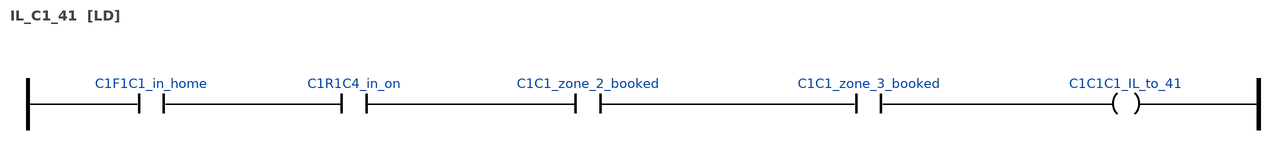
(* LD diagram, written out as Structured Text *)
C1C1C1_IL_to_41 := C1F1C1_in_home AND C1R1C4_in_on AND C1C1_zone_2_booked AND C1C1_zone_3_booked;
END_PROGRAM

PROGRAM IL_C1C2C1_PART_IN_POSITION
  VAR_EXTERNAL
    C1C2_zone_1_booked : BOOL := false;
    C1C2C1_IL_to_part_in_position : BOOL := false;
  END_VAR

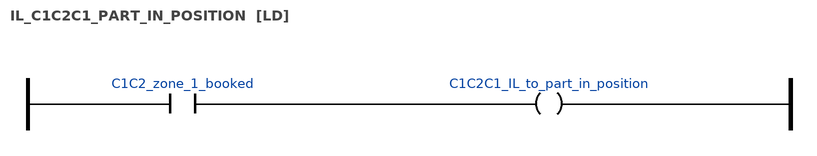
(* LD diagram, written out as Structured Text *)
C1C2C1_IL_to_part_in_position := C1C2_zone_1_booked;
END_PROGRAM

PROGRAM IL_C1C2C1_POSITION_EMPTY
  VAR_EXTERNAL
    C1C2C1_IL_to_part_in_position : BOOL := false;
  END_VAR

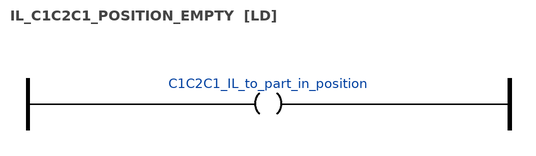
(* LD diagram, written out as Structured Text *)
C1C2C1_IL_to_part_in_position := TRUE;
END_PROGRAM

PROGRAM IL_F1C1_HOME_POS
  VAR_EXTERNAL
    C1F1C2_in_unlocked : BOOL := false;
    C1F1C4_in_off : BOOL := false;
    C1F1C3_in_close : BOOL := false;
    C1F1C4_in_on : BOOL := false;
    Op_24_start : BOOL := false;
    C1F1C3_in_open : BOOL := false;
    C1F1C1_IL_to_home : BOOL := false;
  END_VAR

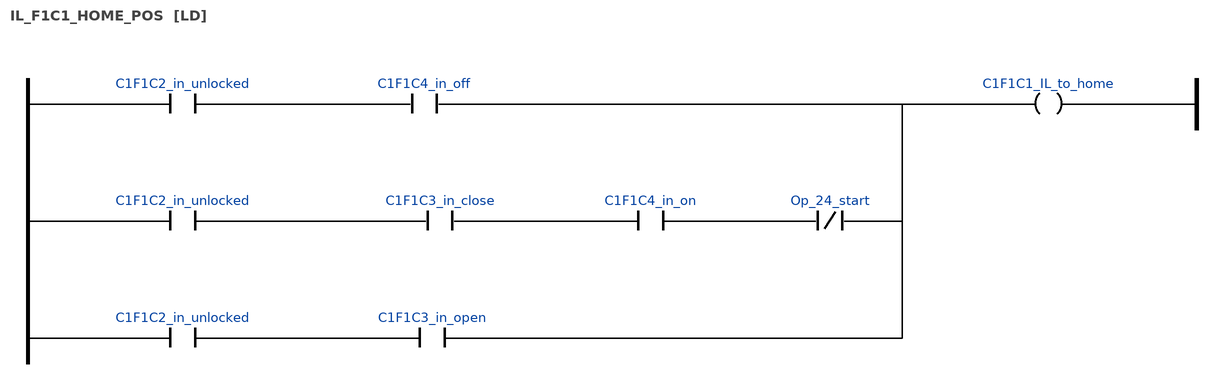
(* LD diagram, written out as Structured Text *)
C1F1C1_IL_to_home := C1F1C2_in_unlocked AND (C1F1C4_in_off OR C1F1C3_in_close AND C1F1C4_in_on AND NOT Op_24_start OR C1F1C3_in_open);
END_PROGRAM

PROGRAM IL_F1C1_WORK_POS
  VAR_EXTERNAL
    C1F1C2_in_unlocked : BOOL := false;
    C1F1C4_in_off : BOOL := false;
    C1F1_zone_2_booked : BOOL := false;
    Op_21_start : BOOL := false;
    Op_21_end : BOOL := false;
    C1F1C4_in_on : BOOL := false;
    C1C1C1_in_empty : BOOL := false;
    C1F1C1_to_work_pos_started : BOOL := false;
    C1F1_zone_3_booked : BOOL := false;
    C1C1C1_in_unprocessed : BOOL := false;
    Op_24_start : BOOL := false;
    C1F1C1_IL_to_work_pos : BOOL := false;
  END_VAR

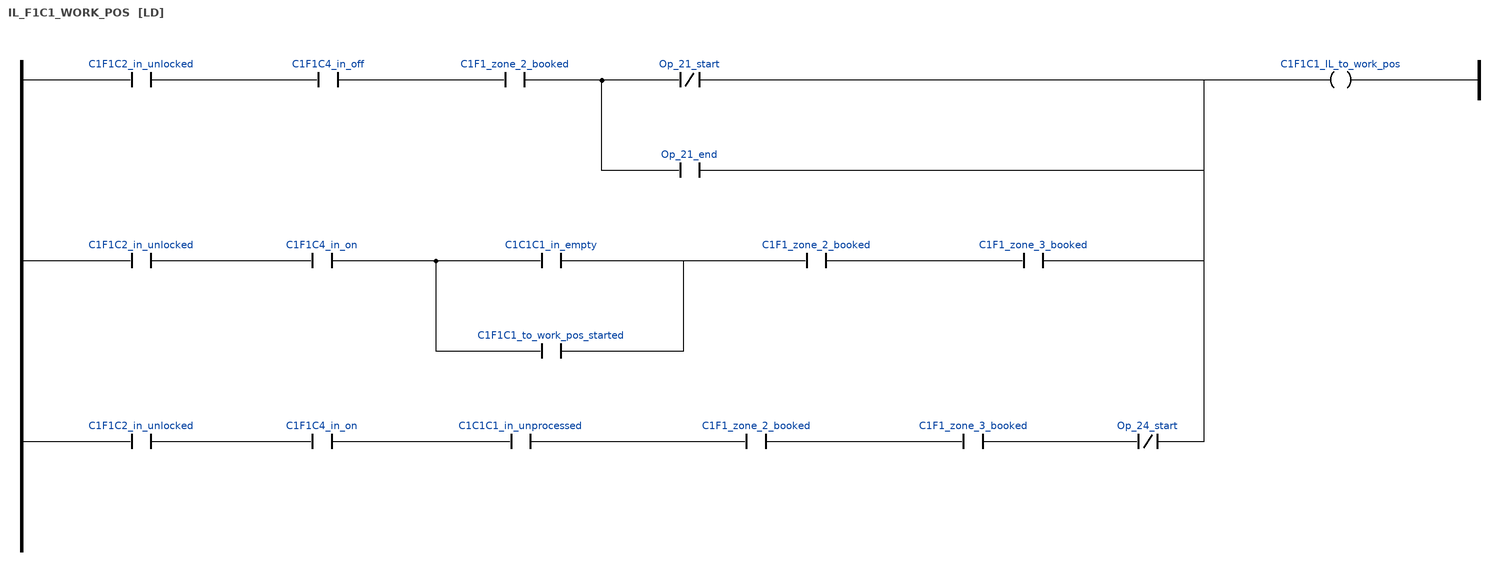
(* LD diagram, written out as Structured Text *)
C1F1C1_IL_to_work_pos := C1F1C2_in_unlocked AND (C1F1C4_in_off AND C1F1_zone_2_booked AND NOT Op_21_start OR C1F1C4_in_off AND C1F1_zone_2_booked AND Op_21_end OR C1F1C4_in_on AND (C1C1C1_in_empty OR C1F1C1_to_work_pos_started) AND C1F1_zone_2_booked AND C1F1_zone_3_booked OR C1F1C4_in_on AND C1C1C1_in_unprocessed AND C1F1_zone_2_booked AND C1F1_zone_3_booked AND NOT Op_24_start);
END_PROGRAM

PROGRAM IL_F1C2_LOCKED
  VAR_EXTERNAL
    C1F1C1_in_home : BOOL := false;
    C1F1C1_in_work_pos : BOOL := false;
    C1F1C2_IL_to_locked : BOOL := false;
  END_VAR

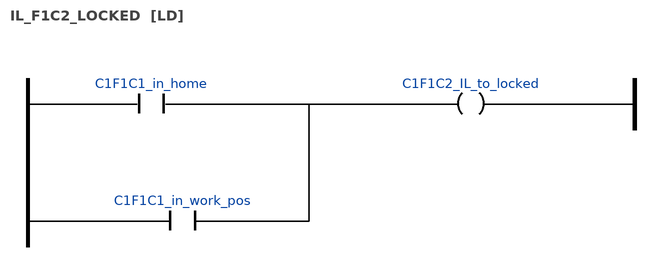
(* LD diagram, written out as Structured Text *)
C1F1C2_IL_to_locked := C1F1C1_in_home OR C1F1C1_in_work_pos;
END_PROGRAM

PROGRAM IL_F1C2_UNLOCKED
  VAR_EXTERNAL
    C1F1C2_IL_to_unlocked : BOOL := false;
  END_VAR

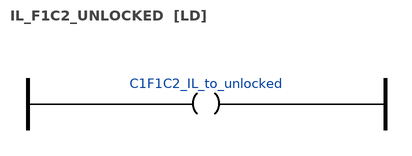
(* LD diagram, written out as Structured Text *)
C1F1C2_IL_to_unlocked := TRUE;
END_PROGRAM

PROGRAM IL_F1C3_CLOSED
  VAR_EXTERNAL
    C1F1C3_IL_to_closed : BOOL := false;
  END_VAR

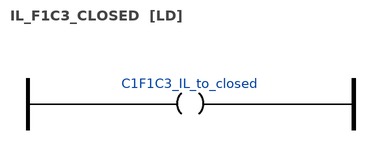
(* LD diagram, written out as Structured Text *)
C1F1C3_IL_to_closed := TRUE;
END_PROGRAM

PROGRAM IL_F1C3_OPEN
  VAR_EXTERNAL
    C1F1C1_in_home : BOOL := false;
    C1F1C1_in_work_pos : BOOL := false;
    C1F1C4_in_off : BOOL := false;
    C1F1C4_in_on : BOOL := false;
    Op_24_start : BOOL := false;
    Op_24_end : BOOL := false;
    C1F1C3_IL_to_open : BOOL := false;
  END_VAR

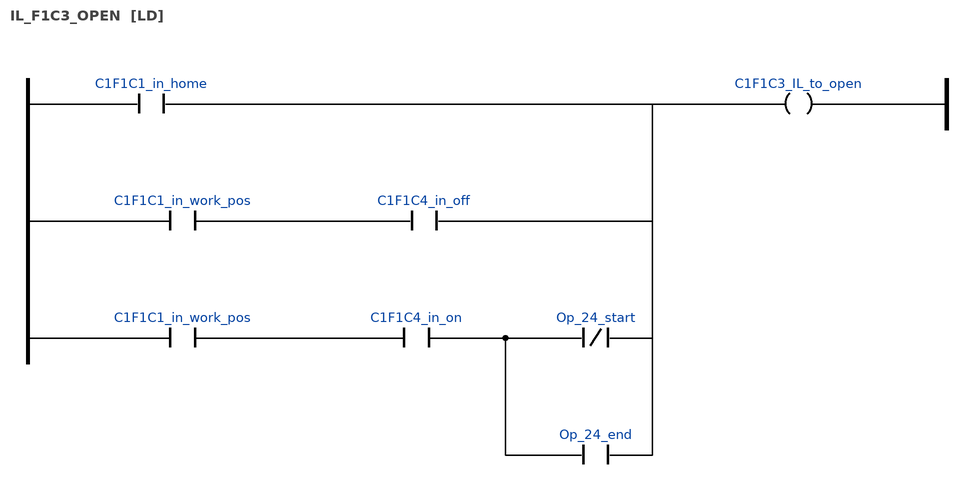
(* LD diagram, written out as Structured Text *)
C1F1C3_IL_to_open := C1F1C1_in_home OR C1F1C1_in_work_pos AND C1F1C4_in_off OR C1F1C1_in_work_pos AND C1F1C4_in_on AND NOT Op_24_start OR C1F1C1_in_work_pos AND C1F1C4_in_on AND Op_24_end;
END_PROGRAM

PROGRAM IL_R1_21
  VAR_EXTERNAL
    C1R1C1_in_open : BOOL := false;
    C1R1C2_in_off : BOOL := false;
    C1C2C1_in_part_in_position : BOOL := false;
    C1R1_zone_1_booked : BOOL := false;
    C1C2C1_in_position_empty : BOOL := false;
    C1R1C1R1_IL_to_21 : BOOL := false;
  END_VAR

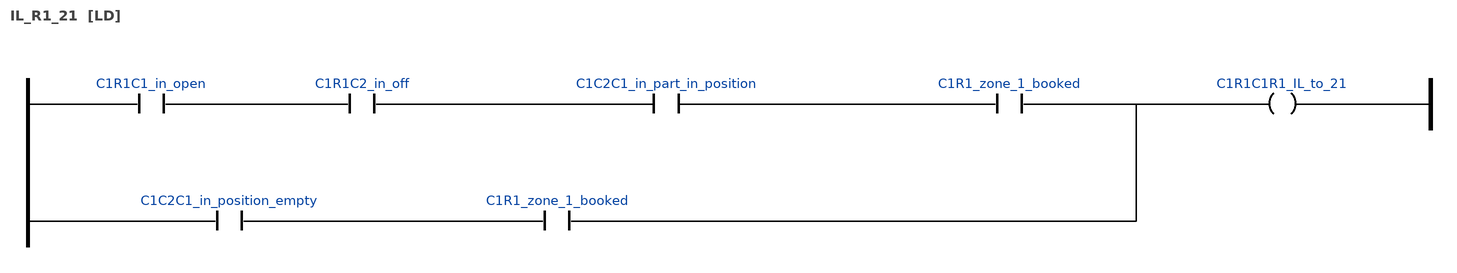
(* LD diagram, written out as Structured Text *)
C1R1C1R1_IL_to_21 := C1R1C1_in_open AND C1R1C2_in_off AND C1C2C1_in_part_in_position AND C1R1_zone_1_booked OR C1C2C1_in_position_empty AND C1R1_zone_1_booked;
END_PROGRAM

PROGRAM IL_R1_22
  VAR_EXTERNAL
    C1F1C1_in_home : BOOL := false;
    C1F1C2_in_locked : BOOL := false;
    C1F1C3_in_open : BOOL := false;
    C1F1C4_in_off : BOOL := false;
    C1R1_Op22_started : BOOL := false;
    C1R1_zone_2_booked : BOOL := false;
    C1R1C1R1_IL_to_22 : BOOL := false;
  END_VAR

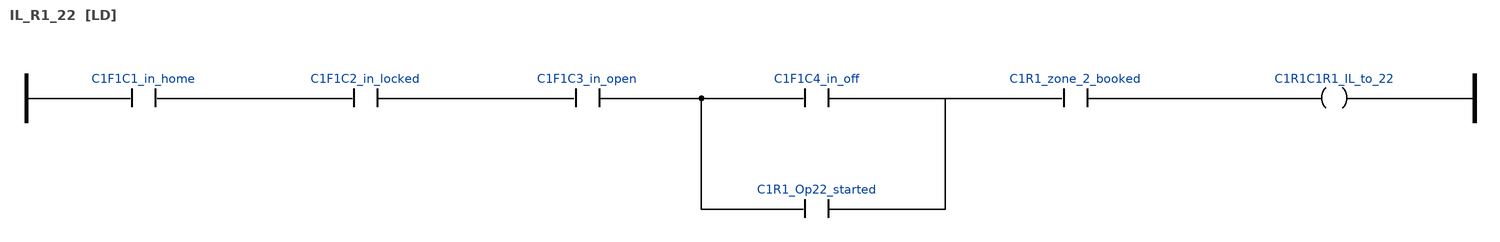
(* LD diagram, written out as Structured Text *)
C1R1C1R1_IL_to_22 := C1F1C1_in_home AND C1F1C2_in_locked AND C1F1C3_in_open AND (C1F1C4_in_off OR C1R1_Op22_started) AND C1R1_zone_2_booked;
END_PROGRAM

PROGRAM IL_R1_23
  VAR_EXTERNAL
    C1R1_zone_2_booked : BOOL := false;
    C1R1C1R1_IL_to_23 : BOOL := false;
  END_VAR

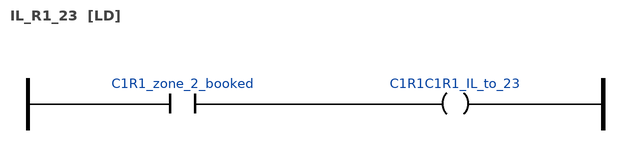
(* LD diagram, written out as Structured Text *)
C1R1C1R1_IL_to_23 := C1R1_zone_2_booked;
END_PROGRAM

PROGRAM IL_R1_24
  VAR_EXTERNAL
    C1C1C1_in_empty : BOOL := false;
    C1F1C1_in_home : BOOL := false;
    C1R1_zone_3_booked : BOOL := false;
    C1C1C1_in_unprocessed : BOOL := false;
    C1F1C1_in_work_pos : BOOL := false;
    C1F1C2_in_locked : BOOL := false;
    C1F1C3_in_open : BOOL := false;
    C1F1C4_in_off : BOOL := false;
    C1F1C3_in_close : BOOL := false;
    C1F1C4_in_on : BOOL := false;
    C1R1C1R1_IL_to_24 : BOOL := false;
  END_VAR

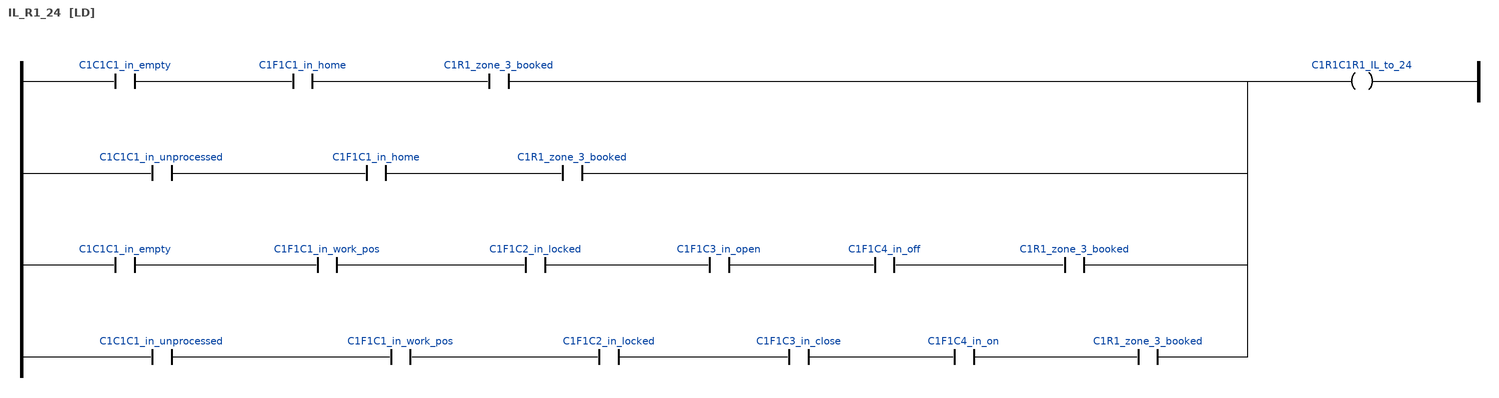
(* LD diagram, written out as Structured Text *)
C1R1C1R1_IL_to_24 := C1C1C1_in_empty AND C1F1C1_in_home AND C1R1_zone_3_booked OR C1C1C1_in_unprocessed AND C1F1C1_in_home AND C1R1_zone_3_booked OR C1C1C1_in_empty AND C1F1C1_in_work_pos AND C1F1C2_in_locked AND C1F1C3_in_open AND C1F1C4_in_off AND C1R1_zone_3_booked OR C1C1C1_in_unprocessed AND C1F1C1_in_work_pos AND C1F1C2_in_locked AND C1F1C3_in_close AND C1F1C4_in_on AND C1R1_zone_3_booked;
END_PROGRAM

PROGRAM CC
  VAR_EXTERNAL
    C1C2C1_in_position_empty : BOOL := false;
    C1C2C2_in_off : BOOL := false;
    C1C2C1_in_part_in_position : BOOL := false;
    C1C2C2_in_on : BOOL := false;
    C1R1_in_inital : BOOL := false;
    C1F1C1_in_home : BOOL := false;
    C1F1C2_in_locked : BOOL := false;
    C1F1C3_in_open : BOOL := false;
    C1F1C4_in_off : BOOL := false;
    C1H1C1_in_normal : BOOL := false;
    CC_B : BOOL := false;
    C1H1C1_in_empty : BOOL := false;
    C1C1C1_in_processed : BOOL := false;
    CC_A : BOOL := false;
    C1_init_position : BOOL := false;
    C1_auto : BOOL := false;
    Start_COPs : BOOL := false;
    COP_C1C1_A_done : BOOL := false;
    COP_C1C2_A_done : BOOL := false;
    COP_C1F1_A_done : BOOL := false;
    COP_C1R1_A_done : BOOL := false;
    All_COP_Done_CC_A : BOOL := false;
    COP_C1C1_B_done : BOOL := false;
    COP_C1C2_B_done : BOOL := false;
    COP_C1F1_B_done : BOOL := false;
    All_COP_Done_CC_B : BOOL := false;
    Op_10_end : BOOL := false;
    Op_11_end : BOOL := false;
    Op_12_end : BOOL := false;
    C1R1_Op20_done : BOOL := false;
    C1R1_Op21_done : BOOL := false;
    C1R1_Op22_done : BOOL := false;
    C1R1_Op23_done : BOOL := false;
    C1R1_Op24_done : BOOL := false;
    Op_30_end : BOOL := false;
    Op_31_end : BOOL := false;
    Op_32_end : BOOL := false;
    Op_33_end : BOOL := false;
    Op_34_end : BOOL := false;
    C1C1_Op40_done : BOOL := false;
    C1C1_Op41_done : BOOL := false;
    C1C1_Op42_done : BOOL := false;
  END_VAR
  VAR  (* added by the conversion: wires and edge detectors of the diagram *)
    _OR45_OUT : BOOL;
  END_VAR

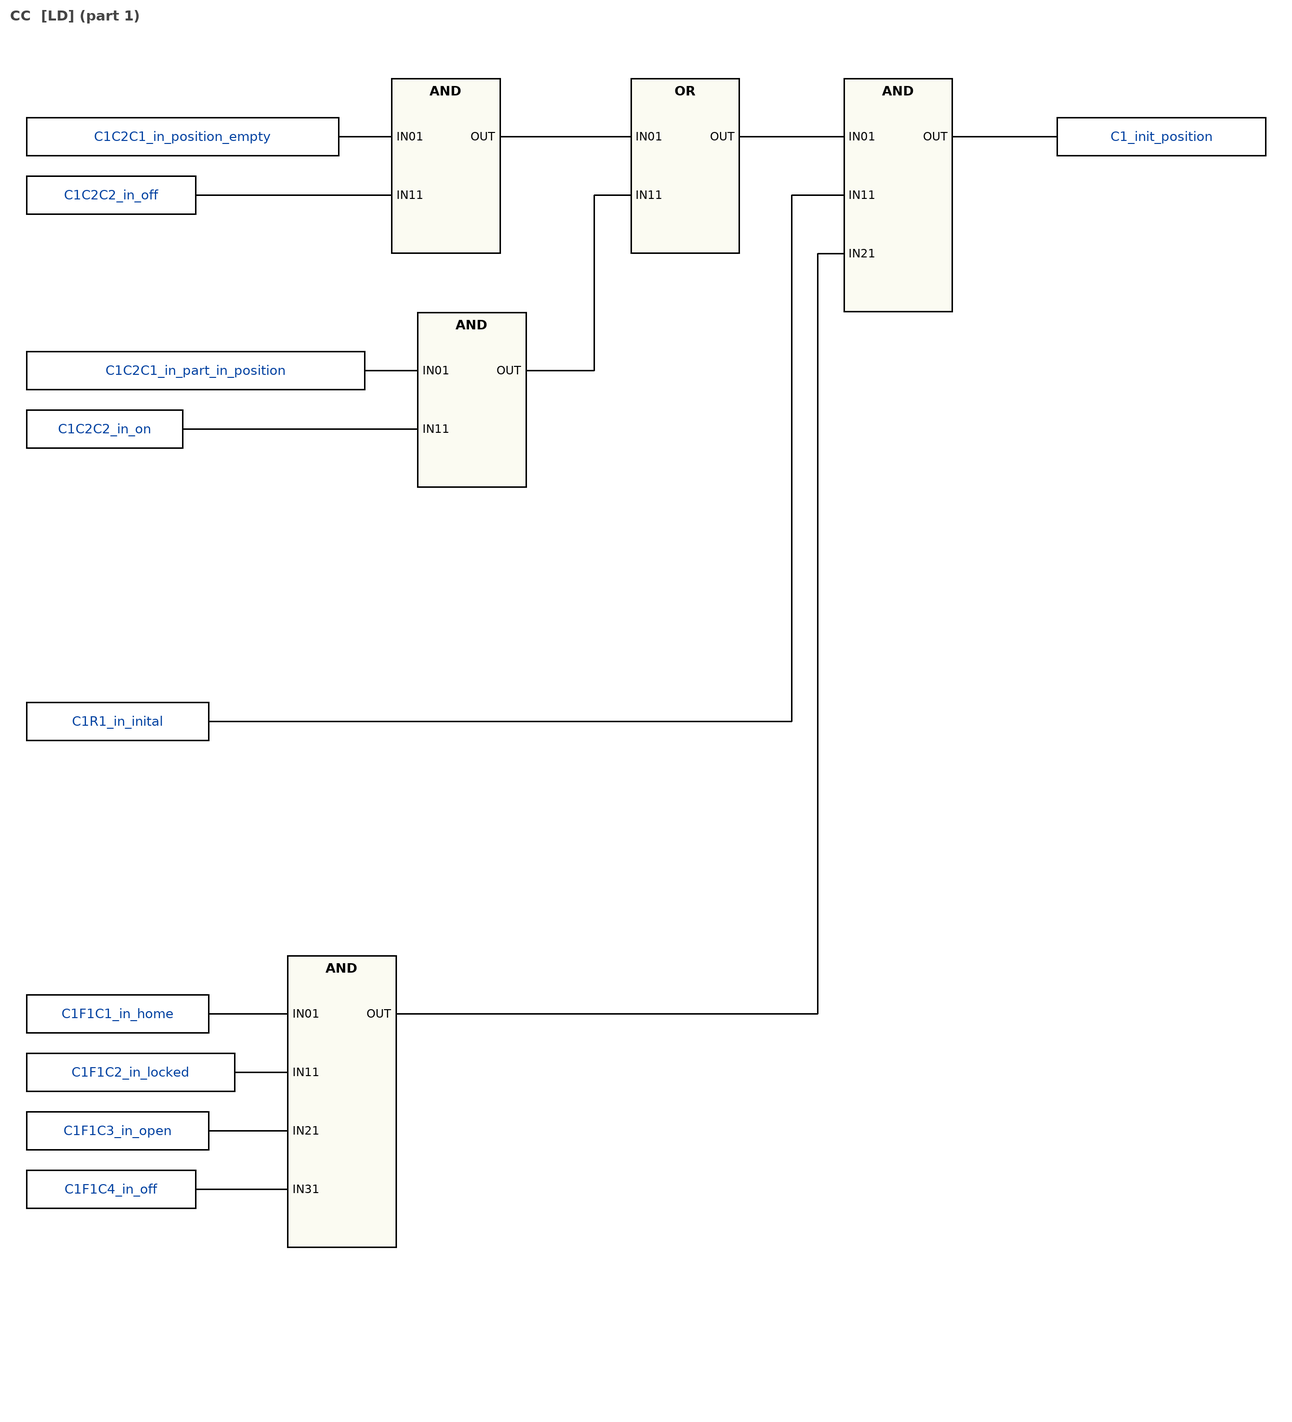
(* LD diagram, written out as Structured Text *)
C1_init_position := (C1C2C1_in_position_empty AND C1C2C2_in_off OR C1C2C1_in_part_in_position AND C1C2C2_in_on) AND C1R1_in_inital AND C1F1C1_in_home AND C1F1C2_in_locked AND C1F1C3_in_open AND C1F1C4_in_off;
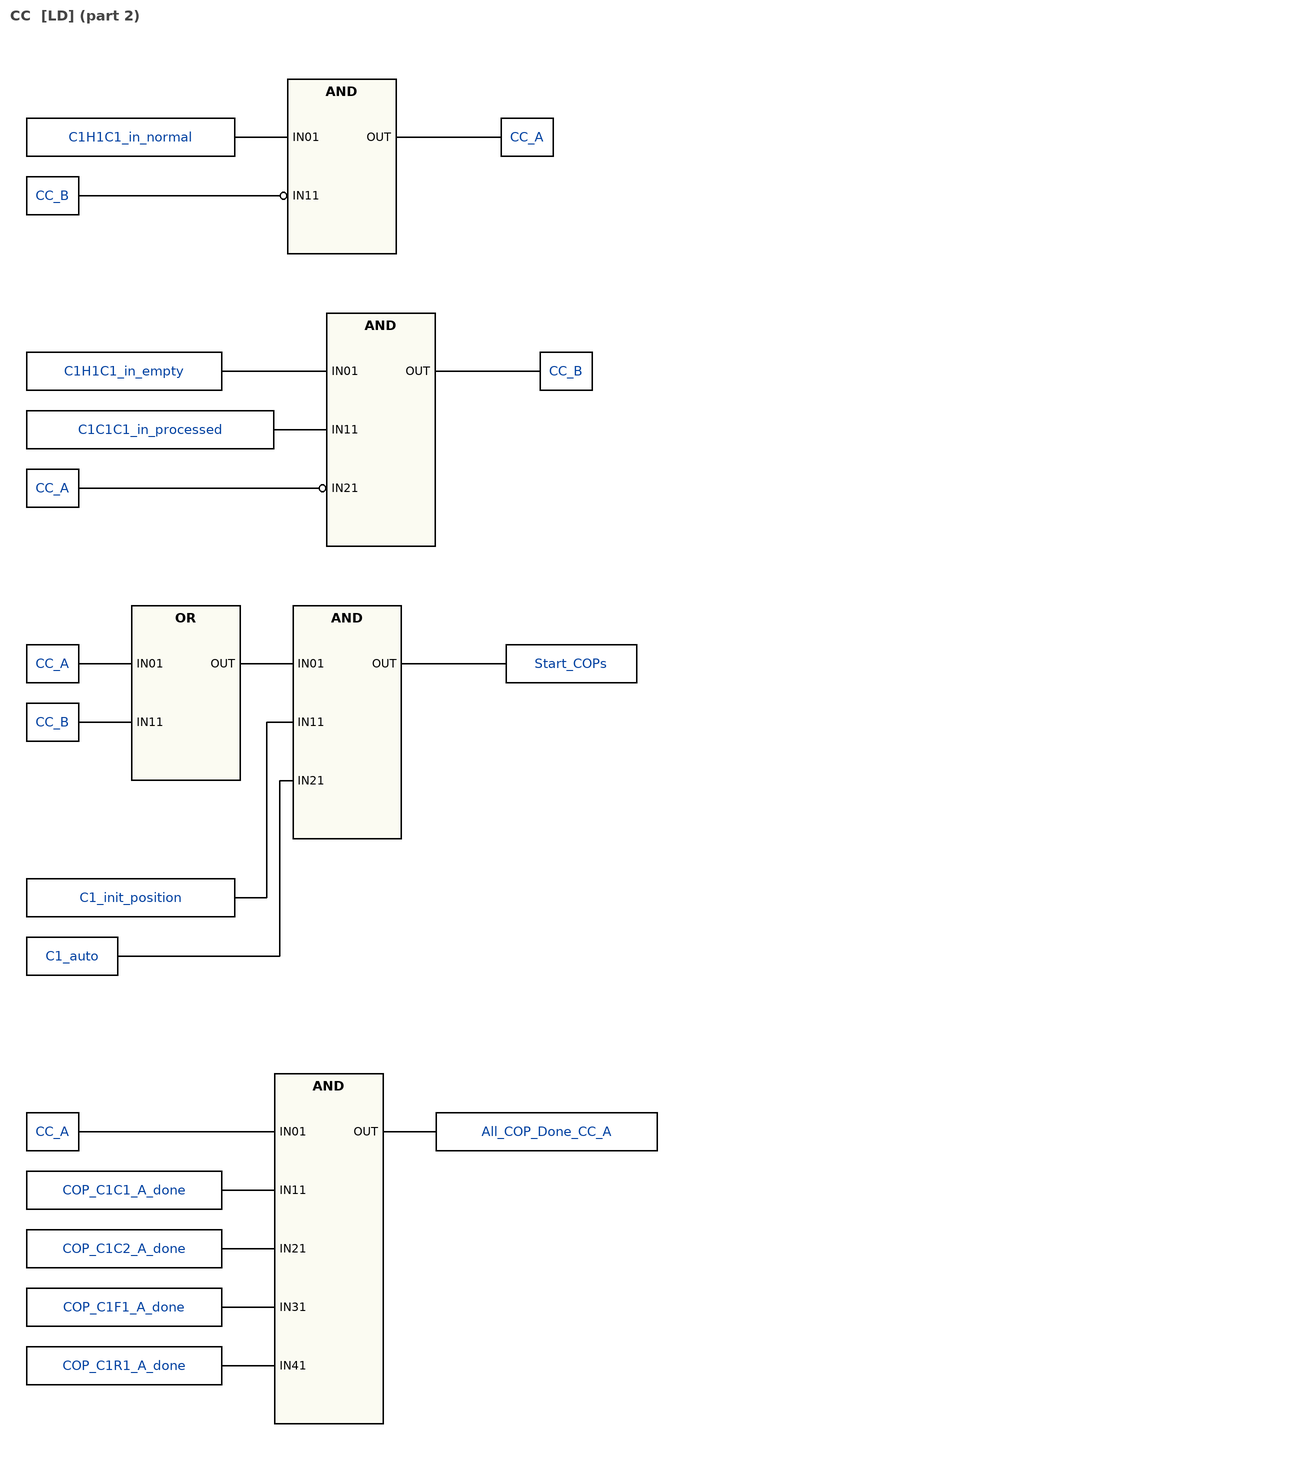
CC_A := C1H1C1_in_normal AND NOT CC_B;
CC_B := C1H1C1_in_empty AND C1C1C1_in_processed AND NOT CC_A;
Start_COPs := (CC_A OR CC_B) AND C1_init_position AND C1_auto;
All_COP_Done_CC_A := CC_A AND COP_C1C1_A_done AND COP_C1C2_A_done AND COP_C1F1_A_done AND COP_C1R1_A_done;
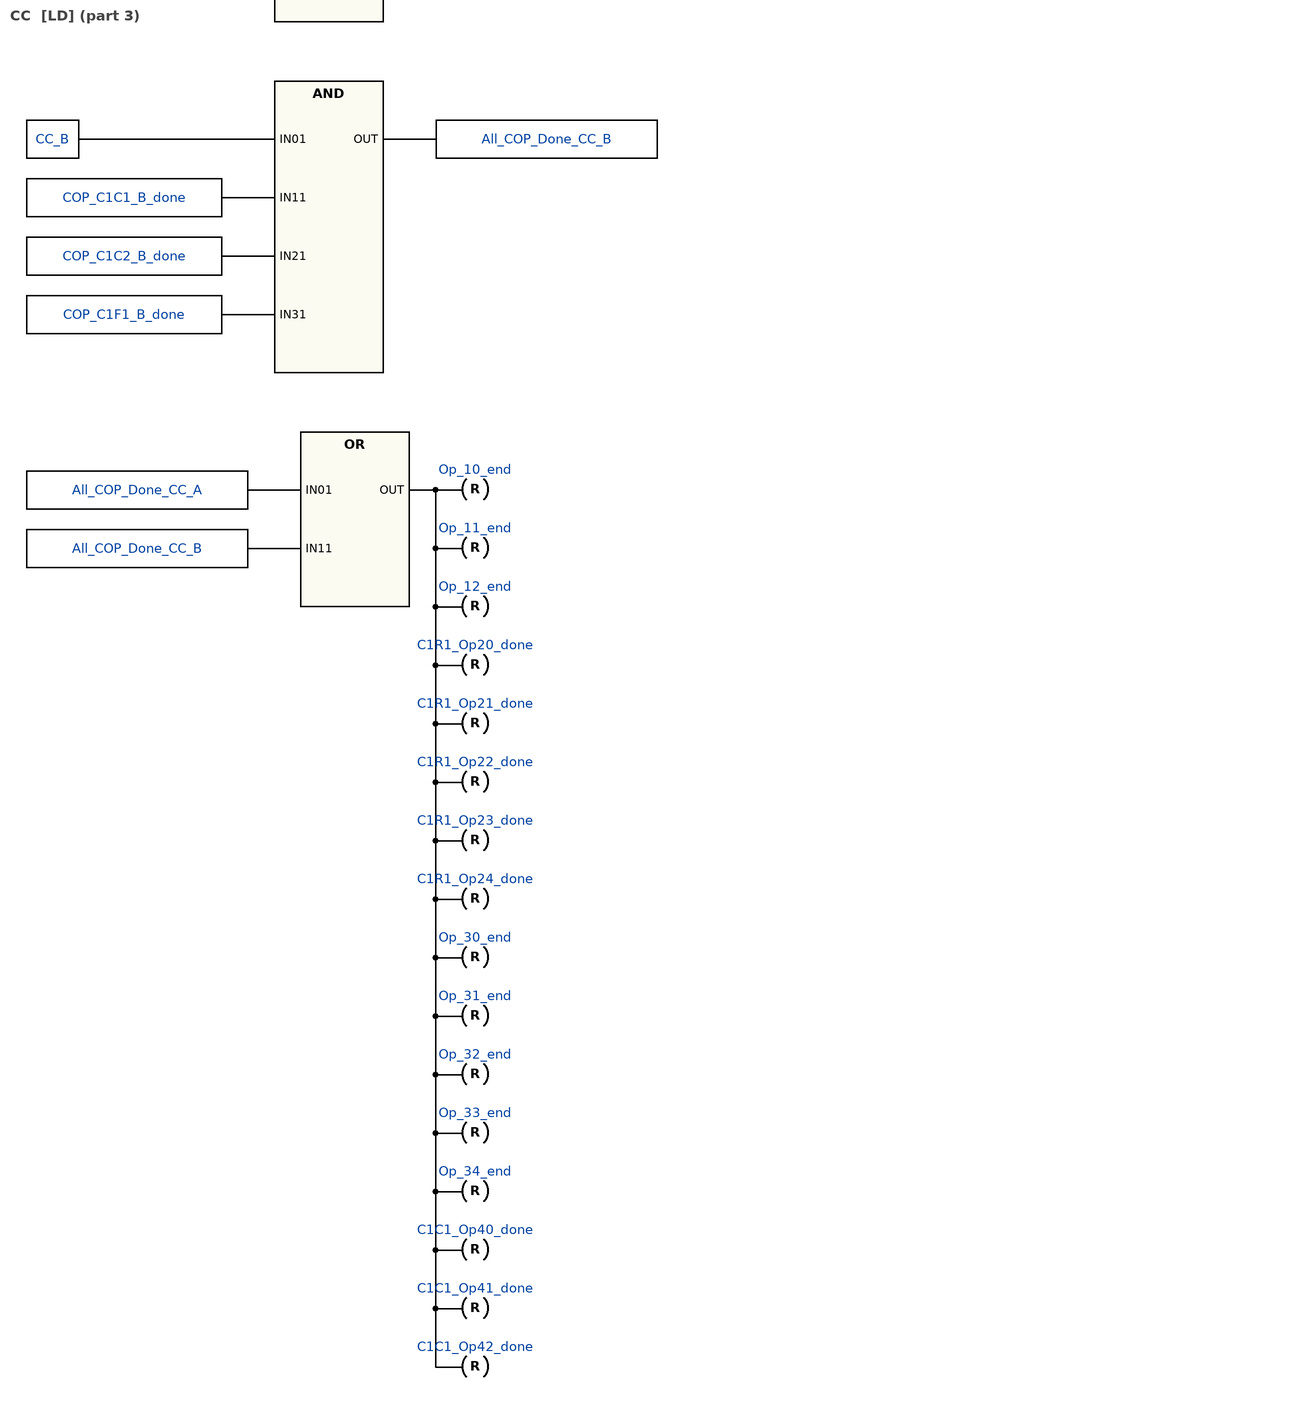
All_COP_Done_CC_B := CC_B AND COP_C1C1_B_done AND COP_C1C2_B_done AND COP_C1F1_B_done;
_OR45_OUT := All_COP_Done_CC_A OR All_COP_Done_CC_B;
IF _OR45_OUT THEN Op_10_end := FALSE; END_IF;
IF _OR45_OUT THEN Op_11_end := FALSE; END_IF;
IF _OR45_OUT THEN Op_12_end := FALSE; END_IF;
IF _OR45_OUT THEN C1R1_Op20_done := FALSE; END_IF;
IF _OR45_OUT THEN C1R1_Op21_done := FALSE; END_IF;
IF _OR45_OUT THEN C1R1_Op22_done := FALSE; END_IF;
IF _OR45_OUT THEN C1R1_Op23_done := FALSE; END_IF;
IF _OR45_OUT THEN C1R1_Op24_done := FALSE; END_IF;
IF _OR45_OUT THEN Op_30_end := FALSE; END_IF;
IF _OR45_OUT THEN Op_31_end := FALSE; END_IF;
IF _OR45_OUT THEN Op_32_end := FALSE; END_IF;
IF _OR45_OUT THEN Op_33_end := FALSE; END_IF;
IF _OR45_OUT THEN Op_34_end := FALSE; END_IF;
IF _OR45_OUT THEN C1C1_Op40_done := FALSE; END_IF;
IF _OR45_OUT THEN C1C1_Op41_done := FALSE; END_IF;
IF _OR45_OUT THEN C1C1_Op42_done := FALSE; END_IF;
END_PROGRAM

CONFIGURATION Example_factory002
  RESOURCE Example_cell002 ON PLC
    VAR_GLOBAL
      Op_10_start : BOOL := false;
      C1C2C1_in_position_empty : BOOL := false;
      C1C2C2_in_off : BOOL := false;
      Op_10_end : BOOL := false;
      C1C2C1_in_part_in_position : BOOL := false;
      C1C2C2_in_on : BOOL := false;
      Op_11_start : BOOL := false;
      TRUE_VAR : BOOL := true;
      C1C2_book_zone_1 : BOOL := false;
      C1C2_zone_1_booked : BOOL := false;
      C1C2C1_goto_part_in_position : BOOL := false;
      C1C2C2_goto_on : BOOL := false;
      C1C2_unbook_zone_1 : BOOL := false;
      Op_11_end : BOOL := false;
      Op_12_start : BOOL := false;
      C1C2C1_goto_position_empty : BOOL := false;
      C1C2C2_goto_off : BOOL := false;
      Op_12_end : BOOL := false;
      C1R1_Op20_exe_start : BOOL := false;
      C1R1_in_inital : BOOL := false;
      C1R1_Op20_exe : BOOL := false;
      C1R1_Op20_done : BOOL := false;
      C1R1_Op21_exe_start : BOOL := false;
      C1R1_book_zone_1 : BOOL := false;
      C1R1_zone_1_booked : BOOL := false;
      C1R1_Op21_exe : BOOL := false;
      C1R1_Op21_done : BOOL := false;
      C1R1_unbook_zone_1 : BOOL := false;
      C1R1_Op22_exe_start : BOOL := false;
      C1R1_Op22_exe : BOOL := false;
      C1R1_Op22_done : BOOL := false;
      C1R1_Op23_exe_start : BOOL := false;
      C1R1_book_zone_2 : BOOL := false;
      C1R1_zone_2_booked : BOOL := false;
      C1R1_Op23_exe : BOOL := false;
      C1R1_Op23_done : BOOL := false;
      C1R1_unbook_zone_2 : BOOL := false;
      C1R1_Op24_exe_start : BOOL := false;
      C1R1_book_zone_3 : BOOL := false;
      C1R1_zone_3_booked : BOOL := false;
      C1R1_Op24_exe : BOOL := false;
      C1R1_Op24_done : BOOL := false;
      C1R1_unbook_zone_3 : BOOL := false;
      Op_30_start : BOOL := false;
      C1F1C1_in_home : BOOL := false;
      C1F1C2_in_locked : BOOL := false;
      C1F1C3_in_open : BOOL := false;
      C1F1C4_in_off : BOOL := false;
      Op_30_end : BOOL := false;
      Op_31_start : BOOL := false;
      Op_31_end : BOOL := false;
      Op_32_start : BOOL := false;
      C1F1C1_goto_home : BOOL := false;
      C1F1C2_goto_locked : BOOL := false;
      C1F1C3_goto_close : BOOL := false;
      C1F1C4_goto_on : BOOL := false;
      C1F1C3_in_close : BOOL := false;
      C1F1C4_in_on : BOOL := false;
      Op_32_end : BOOL := false;
      Op_33_start : BOOL := false;
      C1F1C2_goto_unlocked : BOOL := false;
      C1F1_book_zone_2 : BOOL := false;
      C1F1_book_zone_3 : BOOL := false;
      C1F1C2_in_unlocked : BOOL := false;
      C1F1_zone_2_booked : BOOL := false;
      C1F1_zone_3_booked : BOOL := false;
      C1F1C1_goto_work_pos : BOOL := false;
      C1F1C1_in_work_pos : BOOL := false;
      C1F1_unbook_zone_3 : BOOL := false;
      Op_33_end : BOOL := false;
      Op_34_start : BOOL := false;
      C1F1C3_goto_open : BOOL := false;
      C1F1C4_goto_off : BOOL := false;
      C1F1_unbook_zone_2 : BOOL := false;
      Op_34_end : BOOL := false;
      C1C1_Op40_exe_start : BOOL := false;
      C1C1_Op40_done : BOOL := false;
      C1C1_Op41_exe_start : BOOL := false;
      C1C1_book_zone_2 : BOOL := false;
      C1C1_book_zone_3 : BOOL := false;
      C1C1_zone_2_booked : BOOL := false;
      C1C1_zone_3_booked : BOOL := false;
      C1C1C1_goto_unprocessed : BOOL := false;
      C1C1C1_in_unprocessed : BOOL := false;
      C1C1_unbook_zone_2 : BOOL := false;
      C1C1_unbook_zone_3 : BOOL := false;
      C1C1_Op41_done : BOOL := false;
      C1C1_Op42_exe_start : BOOL := false;
      C1C1C1_goto_processed : BOOL := false;
      C1C1C1_in_processed : BOOL := false;
      C1C1_Op42_done : BOOL := false;
      Start_COPs : BOOL := false;
      CC_A : BOOL := false;
      COP_C1C1_A_done : BOOL := false;
      All_COP_Done_CC_A : BOOL := false;
      CC_B : BOOL := false;
      C1C1_Op43_exe_start : BOOL := false;
      C1C1_Op43_done : BOOL := false;
      COP_C1C1_B_done : BOOL := false;
      All_COP_Done_CC_B : BOOL := false;
      COP_C1C2_A_done : BOOL := false;
      COP_C1C2_B_done : BOOL := false;
      COP_C1F1_A_done : BOOL := false;
      COP_C1F1_B_done : BOOL := false;
      COP_C1R1_A_done : BOOL := false;
      C1R1_Op20_IL : BOOL := false;
      C1R1_Op20_started : BOOL := false;
      C1R1_Op21_IL : BOOL := false;
      C1R1_Op21_started : BOOL := false;
      C1R1_Op22_IL : BOOL := false;
      C1R1_Op22_started : BOOL := false;
      C1R1_Op23_IL : BOOL := false;
      C1R1_Op23_started : BOOL := false;
      C1R1_Op24_IL : BOOL := false;
      C1R1_Op24_started : BOOL := false;
      C1R1_ext_lb_0 : BOOL := false;
      C1R1_ext_Ob_0 : BOOL := false;
      C1R1_ext_lb_1 : BOOL := false;
      C1R1_ext_Ob_1 : BOOL := false;
      C1R1_ext_lb_2 : BOOL := false;
      C1R1_ext_Ob_2 : BOOL := false;
      C1R1_ext_lb_3 : BOOL := false;
      C1R1_ext_Ob_3 : BOOL := false;
      C1R1_ext_lb_4 : BOOL := false;
      C1R1_ext_Ob_4 : BOOL := false;
      C1R1_ext_lb_5 : BOOL := false;
      C1R1_ext_Ob_5 : BOOL := false;
      C1R1_ext_lb_6 : BOOL := false;
      C1R1_ext_Ob_6 : BOOL := false;
      C1R1_ext_lb_7 : BOOL := false;
      C1R1_ext_Ob_7 : BOOL := false;
      C1R1_ext_machine_OK : BOOL := false;
      C1R1_IL_OK : BOOL := false;
      C1C1_Op40_exe : BOOL := false;
      C1C1_Op40_IL : BOOL := false;
      C1C1_Op40_started : BOOL := false;
      C1C1_Op41_exe : BOOL := false;
      C1C1_Op41_IL : BOOL := false;
      C1C1_Op41_started : BOOL := false;
      C1C1_Op42_exe : BOOL := false;
      C1C1_Op42_IL : BOOL := false;
      C1C1_Op42_started : BOOL := false;
      C1C1_Op43_exe : BOOL := false;
      C1C1_Op43_IL : BOOL := false;
      C1C1_Op43_started : BOOL := false;
      C1C1_ext_lb_0 : BOOL := false;
      C1C1_ext_Ob_0 : BOOL := false;
      C1C1_ext_lb_1 : BOOL := false;
      C1C1_ext_Ob_1 : BOOL := false;
      C1C1_ext_lb_2 : BOOL := false;
      C1C1_ext_Ob_2 : BOOL := false;
      C1C1_ext_lb_3 : BOOL := false;
      C1C1_ext_Ob_3 : BOOL := false;
      C1C1_ext_lb_4 : BOOL := false;
      C1C1_ext_Ob_4 : BOOL := false;
      C1C1_ext_lb_5 : BOOL := false;
      C1C1_ext_Ob_5 : BOOL := false;
      C1C1_ext_lb_6 : BOOL := false;
      C1C1_ext_Ob_6 : BOOL := false;
      C1C1_ext_lb_7 : BOOL := false;
      C1C1_ext_Ob_7 : BOOL := false;
      C1C1_ext_machine_OK : BOOL := false;
      C1C1_IL_OK : BOOL := false;
      C1C2C1_IL_to_part_in_position : BOOL := false;
      C1C2C1_to_part_in_position_started : BOOL := false;
      C1C2C1_QS1 : BOOL := false;
      C1C2C1_IL_to_position_empty : BOOL := false;
      C1C2C1_to_position_empty_started : BOOL := false;
      C1C2C1_QS2 : BOOL := false;
      Not_Connected : BOOL := false;
      C1F1C1_IL_to_home : BOOL := false;
      C1F1C1_to_home_started : BOOL := false;
      C1F1C1_QS1 : BOOL := false;
      C1F1C1_IS1 : BOOL := false;
      C1F1C1_IL_to_work_pos : BOOL := false;
      C1F1C1_to_work_pos_started : BOOL := false;
      C1F1C1_QS2 : BOOL := false;
      C1F1C1_IS2 : BOOL := false;
      C1F1C2_IL_to_locked : BOOL := false;
      C1F1C2_to_locked_started : BOOL := false;
      C1F1C2_QS1 : BOOL := false;
      C1F1C2_IS1 : BOOL := false;
      C1F1C2_IL_to_unlocked : BOOL := false;
      C1F1C2_to_unlocked_started : BOOL := false;
      C1F1C2_QS2 : BOOL := false;
      C1F1C2_IS2 : BOOL := false;
      C1F1C3_IL_to_open : BOOL := false;
      C1F1C3_to_open_started : BOOL := false;
      C1F1C3_QS1 : BOOL := false;
      C1F1C3_IS1A : BOOL := false;
      C1F1C3_IS1B : BOOL := false;
      C1F1C3_IL_to_close : BOOL := false;
      C1F1C3_to_close_started : BOOL := false;
      C1F1C3_QS2 : BOOL := false;
      C1F1C3_IS2A : BOOL := false;
      C1F1C3_IS2B : BOOL := false;
      C1F1C4_IS2A : BOOL := false;
      C1F1C4_IS2B : BOOL := false;
      C1R1C4_in_on : BOOL := false;
      C1C1C1_IL_to_41 : BOOL := false;
      Op_24_start : BOOL := false;
      Op_21_start : BOOL := false;
      Op_21_end : BOOL := false;
      C1C1C1_in_empty : BOOL := false;
      C1F1C3_IL_to_closed : BOOL := false;
      Op_24_end : BOOL := false;
      C1R1C1_in_open : BOOL := false;
      C1R1C2_in_off : BOOL := false;
      C1R1C1R1_IL_to_21 : BOOL := false;
      C1R1C1R1_IL_to_22 : BOOL := false;
      C1R1C1R1_IL_to_23 : BOOL := false;
      C1R1C1R1_IL_to_24 : BOOL := false;
      C1H1C1_in_normal : BOOL := false;
      C1H1C1_in_empty : BOOL := false;
      C1_init_position : BOOL := false;
      C1_auto : BOOL := false;
    END_VAR
    VAR_GLOBAL CONSTANT
      Constant_20 : INT := 20;
      Constant_21 : INT := 21;
      Constant_22 : INT := 22;
      Constant_23 : INT := 23;
      Constant_24 : INT := 24;
      Constant_40 : INT := 40;
      Constant_41 : INT := 41;
      Constant_42 : INT := 42;
      Constant_43 : INT := 43;
    END_VAR
    TASK Task_EOP10_a(PRIORITY := 0);
    TASK Task_EOP10_b(PRIORITY := 0);
    TASK Task_EOP11(PRIORITY := 0);
    TASK Task_EOP12(PRIORITY := 0);
    TASK Task_EOP20(PRIORITY := 0);
    TASK Task_EOP21(PRIORITY := 0);
    TASK Task_EOP22(PRIORITY := 0);
    TASK Task_EOP23(PRIORITY := 0);
    TASK Task_EOP24(PRIORITY := 0);
    TASK Task_EOP30(PRIORITY := 0);
    TASK Task_EOP31(PRIORITY := 0);
    TASK Task_EOP32(PRIORITY := 0);
    TASK Task_EOP33(PRIORITY := 0);
    TASK Task_EOP34(PRIORITY := 0);
    TASK Task_EOP40(PRIORITY := 0);
    TASK Task_EOP41(PRIORITY := 0);
    TASK Task_EOP42(PRIORITY := 0);
    TASK Task_COP_C1C1_A(PRIORITY := 0);
    TASK Task_COP_C1C1_B(PRIORITY := 0);
    TASK Task_COP_C1C2_A(PRIORITY := 0);
    TASK Task_COP_C1C2_B(PRIORITY := 0);
    TASK Task_COP_C1F1_A(PRIORITY := 0);
    TASK Task_COP_C1F1_B(PRIORITY := 0);
    TASK Task_COP_C1R1_A(PRIORITY := 0);
    TASK Task_FB_C1R1_External_Machine_comm_-_5_OP(PRIORITY := 0);
    TASK Task_FB_C1C1_External_Machine_comm_-_4_OP(PRIORITY := 0);
    TASK Task_FB_C1C2C1_Belt_Conveyor(PRIORITY := 0);
    TASK Task_FB_C1F1C1_Two_Position_Movement(PRIORITY := 0);
    TASK Task_FB_C1F1C2_Two_Position_Movement(PRIORITY := 0);
    TASK Task_FB_C1F1C3_Two_Position_Movement(PRIORITY := 0);
    TASK Task_FB_C1F1C4_Part_Detection_x2(PRIORITY := 0);
    TASK Task_FB_Zone_1(PRIORITY := 0);
    TASK Task_FB_Zone_2(PRIORITY := 0);
    TASK Task_FB_Zone_3(PRIORITY := 0);
    TASK Task_IL_C1_41(PRIORITY := 0);
    TASK Task_IL_C1C2C1_PART_IN_POSITION(PRIORITY := 0);
    TASK Task_IL_C1C2C1_POSITION_EMPTY(PRIORITY := 0);
    TASK Task_IL_F1C1_HOME_POS(PRIORITY := 0);
    TASK Task_IL_F1C1_WORK_POS(PRIORITY := 0);
    TASK Task_IL_F1C2_LOCKED(PRIORITY := 0);
    TASK Task_IL_F1C2_UNLOCKED(PRIORITY := 0);
    TASK Task_IL_F1C3_CLOSED(PRIORITY := 0);
    TASK Task_IL_F1C3_OPEN(PRIORITY := 0);
    TASK Task_IL_R1_21(PRIORITY := 0);
    TASK Task_IL_R1_22(PRIORITY := 0);
    TASK Task_IL_R1_23(PRIORITY := 0);
    TASK Task_IL_R1_24(PRIORITY := 0);
    TASK Task_CC(PRIORITY := 0);
    PROGRAM InstanceOf_EOP10_a WITH Task_EOP10_a : EOP10_a;
    PROGRAM InstanceOf_EOP10_b WITH Task_EOP10_b : EOP10_b;
    PROGRAM InstanceOf_EOP11 WITH Task_EOP11 : EOP11;
    PROGRAM InstanceOf_EOP12 WITH Task_EOP12 : EOP12;
    PROGRAM InstanceOf_EOP20 WITH Task_EOP20 : EOP20;
    PROGRAM InstanceOf_EOP21 WITH Task_EOP21 : EOP21;
    PROGRAM InstanceOf_EOP22 WITH Task_EOP22 : EOP22;
    PROGRAM InstanceOf_EOP23 WITH Task_EOP23 : EOP23;
    PROGRAM InstanceOf_EOP24 WITH Task_EOP24 : EOP24;
    PROGRAM InstanceOf_EOP30 WITH Task_EOP30 : EOP30;
    PROGRAM InstanceOf_EOP31 WITH Task_EOP31 : EOP31;
    PROGRAM InstanceOf_EOP32 WITH Task_EOP32 : EOP32;
    PROGRAM InstanceOf_EOP33 WITH Task_EOP33 : EOP33;
    PROGRAM InstanceOf_EOP34 WITH Task_EOP34 : EOP34;
    PROGRAM InstanceOf_EOP40 WITH Task_EOP40 : EOP40;
    PROGRAM InstanceOf_EOP41 WITH Task_EOP41 : EOP41;
    PROGRAM InstanceOf_EOP42 WITH Task_EOP42 : EOP42;
    PROGRAM InstanceOf_COP_C1C1_A WITH Task_COP_C1C1_A : COP_C1C1_A;
    PROGRAM InstanceOf_COP_C1C1_B WITH Task_COP_C1C1_B : COP_C1C1_B;
    PROGRAM InstanceOf_COP_C1C2_A WITH Task_COP_C1C2_A : COP_C1C2_A;
    PROGRAM InstanceOf_COP_C1C2_B WITH Task_COP_C1C2_B : COP_C1C2_B;
    PROGRAM InstanceOf_COP_C1F1_A WITH Task_COP_C1F1_A : COP_C1F1_A;
    PROGRAM InstanceOf_COP_C1F1_B WITH Task_COP_C1F1_B : COP_C1F1_B;
    PROGRAM InstanceOf_COP_C1R1_A WITH Task_COP_C1R1_A : COP_C1R1_A;
    PROGRAM InstanceOf_FB_C1R1_External_Machine_comm_-_5_OP WITH Task_FB_C1R1_External_Machine_comm_-_5_OP : FB_C1R1_External_Machine_comm_-_5_OP;
    PROGRAM InstanceOf_FB_C1C1_External_Machine_comm_-_4_OP WITH Task_FB_C1C1_External_Machine_comm_-_4_OP : FB_C1C1_External_Machine_comm_-_4_OP;
    PROGRAM InstanceOf_FB_C1C2C1_Belt_Conveyor WITH Task_FB_C1C2C1_Belt_Conveyor : FB_C1C2C1_Belt_Conveyor;
    PROGRAM InstanceOf_FB_C1F1C1_Two_Position_Movement WITH Task_FB_C1F1C1_Two_Position_Movement : FB_C1F1C1_Two_Position_Movement;
    PROGRAM InstanceOf_FB_C1F1C2_Two_Position_Movement WITH Task_FB_C1F1C2_Two_Position_Movement : FB_C1F1C2_Two_Position_Movement;
    PROGRAM InstanceOf_FB_C1F1C3_Two_Position_Movement WITH Task_FB_C1F1C3_Two_Position_Movement : FB_C1F1C3_Two_Position_Movement;
    PROGRAM InstanceOf_FB_C1F1C4_Part_Detection_x2 WITH Task_FB_C1F1C4_Part_Detection_x2 : FB_C1F1C4_Part_Detection_x2;
    PROGRAM InstanceOf_FB_Zone_1 WITH Task_FB_Zone_1 : FB_Zone_1;
    PROGRAM InstanceOf_FB_Zone_2 WITH Task_FB_Zone_2 : FB_Zone_2;
    PROGRAM InstanceOf_FB_Zone_3 WITH Task_FB_Zone_3 : FB_Zone_3;
    PROGRAM InstanceOf_IL_C1_41 WITH Task_IL_C1_41 : IL_C1_41;
    PROGRAM InstanceOf_IL_C1C2C1_PART_IN_POSITION WITH Task_IL_C1C2C1_PART_IN_POSITION : IL_C1C2C1_PART_IN_POSITION;
    PROGRAM InstanceOf_IL_C1C2C1_POSITION_EMPTY WITH Task_IL_C1C2C1_POSITION_EMPTY : IL_C1C2C1_POSITION_EMPTY;
    PROGRAM InstanceOf_IL_F1C1_HOME_POS WITH Task_IL_F1C1_HOME_POS : IL_F1C1_HOME_POS;
    PROGRAM InstanceOf_IL_F1C1_WORK_POS WITH Task_IL_F1C1_WORK_POS : IL_F1C1_WORK_POS;
    PROGRAM InstanceOf_IL_F1C2_LOCKED WITH Task_IL_F1C2_LOCKED : IL_F1C2_LOCKED;
    PROGRAM InstanceOf_IL_F1C2_UNLOCKED WITH Task_IL_F1C2_UNLOCKED : IL_F1C2_UNLOCKED;
    PROGRAM InstanceOf_IL_F1C3_CLOSED WITH Task_IL_F1C3_CLOSED : IL_F1C3_CLOSED;
    PROGRAM InstanceOf_IL_F1C3_OPEN WITH Task_IL_F1C3_OPEN : IL_F1C3_OPEN;
    PROGRAM InstanceOf_IL_R1_21 WITH Task_IL_R1_21 : IL_R1_21;
    PROGRAM InstanceOf_IL_R1_22 WITH Task_IL_R1_22 : IL_R1_22;
    PROGRAM InstanceOf_IL_R1_23 WITH Task_IL_R1_23 : IL_R1_23;
    PROGRAM InstanceOf_IL_R1_24 WITH Task_IL_R1_24 : IL_R1_24;
    PROGRAM InstanceOf_CC WITH Task_CC : CC;
  END_RESOURCE
END_CONFIGURATION
